TYPE ST_CtrlOutFunctionForks :
STRUCT
	ForkInCenter		: BOOL;
	MotionRunning		: BOOL; //fork motion running
END_STRUCT
END_TYPE

(* stored: Version 1.1.0.1, ProductVersion 3.1.4024.9
   DUT ST_CtrlOutFunctionForks: Id {a4f5952e-969d-4ca4-819f-60cc3220f050} *)
